(* PLC project  *)

CONFIGURATION Extra
END_CONFIGURATION
